TYPE ST_IO :
STRUCT
	sName			: STRING		;
	iState			: E_State		;
	xState			: REFERENCE TO BOOL 			;
	xStateHMI		: BOOL 			;
	xInvisible		: BOOL			;
	
END_STRUCT
END_TYPE

(* stored: Version 1.1.0.1, ProductVersion 3.1.4024.12
   DUT ST_IO: Id {a61a3b47-3ba0-4596-ba00-dae427afc65a} *)
